Fanuc KAREL source: CA0115.KL

-- PROVISIONAL review KL for V1013-1; original PC SHA256 c4e46bd1b2dc9679f86627cb91ce68c8857303c15ff2e71e103afa4bf6894d37
-- Incomplete behavior may be omitted. Consult companion uncertainty JSON. Do not deploy.
PROGRAM CA0115
%NOLOCKGROUP
BEGIN
  -- UNRESOLVED_PC offsets 0-1; opcodes 7B
  -- UNRESOLVED_PC offsets 6-16; opcodes 2D,7F
  -- UNRESOLVED_PC offsets 21-25; opcodes 7F
  -- UNRESOLVED_PC offsets 30-37; opcodes 9C,23
  -- UNRESOLVED_PC offsets 42-49; opcodes 9D,23
  -- UNRESOLVED_PC offsets 54-65; opcodes 2E,23
  -- UNRESOLVED_PC offsets 70-77; opcodes 9D,23
  -- UNRESOLVED_PC offsets 82-91; opcodes 3F,75
  -- UNRESOLVED_PC offsets 96-110; opcodes 2E,22,9D,33,35
  -- UNRESOLVED_PC offsets 115-129; opcodes 2E,22,9D,33,35
  -- UNRESOLVED_PC offsets 134-149; opcodes 2E,22,32,35
  -- UNRESOLVED_PC offsets 154-169; opcodes 2E,22,32,35
  -- UNRESOLVED_PC offsets 174-280; opcodes 27,22,22,22,22,22,22,22,22,22,22,22,22,22,22,22,22,AA,23
  -- UNRESOLVED_PC offsets 285-289; opcodes 7F
END CA0115
